TYPE ST_TapCmd :
STRUCT
	OnOff: BOOL;
END_STRUCT
END_TYPE

(* stored: Version 1.1.0.1, ProductVersion 3.1.4024.12
   DUT ST_TapCmd: Id {417530f1-d41c-452e-b9e8-4abea7d7aa05} *)
